Staubli VAL3: IsDigtal.pgx

program IsDigtal(num x_nIOid (dimensions=1), bool& x_bRes (dimensions=1))
begin
  x_bRes=x_nIOid<=134

end
